FUNCTION TryConvert_UDINT_TO_LREAL : BOOL
VAR_INPUT
	in : UDINT;
	out : REFERENCE TO LREAL;
END_VAR

out := UDINT_TO_LREAL(in);
TryConvert_UDINT_TO_LREAL := TRUE;

END_FUNCTION

(* stored: Version 1.1.0.1, ProductVersion 3.1.4024.12
   POU TryConvert_UDINT_TO_LREAL: Id {760459b9-49f5-4d08-9992-cc84fc6b9c58}, SpecialFunc None *)
